// TIA Portal V20 export
TYPE "AnalogInAction_DT"
   STRUCT
      BadPartOnFixture { ExternalVisible := 'False'} : Bool;
      ID_Measure : Int;
   END_STRUCT;
END_TYPE
